# EPICS substitutions: ek9000App/Db/EL3044.substitutions
file EL3044.template
{       pattern
        {
                TERMINAL,

        }
        {
        }
}
